// TIA Portal V17 export
// export: Created 2024-01-30T08:49:12.6809505Z, ExportSetting WithDefaults, DisplayName Totally Integrated Automation Portal, DisplayVersion V17 Update 6, DisplayName TIA Portal Openness, DisplayVersion V17 Update 6, DisplayName TIA Portal Version Control Interface, DisplayVersion V17, DisplayName STEP 7 Professional, DisplayVersion V17 Update 6, DisplayName STEP 7 Safety, DisplayVersion V17 Update 6, DisplayName WinCC Advanced, DisplayVersion V17 Update 6
FUNCTION_BLOCK "MeasTable_SQ"   // FB15, GRAPH
AUTHOR : an38503
VERSION : 0.1
// stored: AcknowledgeErrorsRequired true, AutoNumber true, GraphVersion 6.0, InitialValuesAcquisition false, IsIECCheckEnabled false, LanguageInNetworks FBD, LockOperatingMode false, PermanentILProcessingInMANMode false, SetENOAutomatically false, SkipSteps false, UDAEnableTagReadback false, WithAlarmHandling true
   // inherited from GRAPH_BASE
   VAR
      OFF_SQ_BASE : Bool;
   END_VAR
   VAR_INPUT
      OFF_SQ { ExternalAccessible := 'False'; ExternalVisible := 'False'; ExternalWritable := 'False'} : Bool := false;   // Kette ausschalten
      INIT_SQ { ExternalAccessible := 'False'; ExternalVisible := 'False'; ExternalWritable := 'False'} : Bool := false;   // Kette in Initialzustand versetzen
      ACK_EF { ExternalAccessible := 'False'; ExternalVisible := 'False'; ExternalWritable := 'False'} : Bool := false;   // Alle Fehler und Störungen quittieren
      S_PREV { ExternalAccessible := 'False'; ExternalVisible := 'False'; ExternalWritable := 'False'} : Bool := false;   // Vorherigen Schritt am Parameter S_NO ausgeben
      S_NEXT { ExternalAccessible := 'False'; ExternalVisible := 'False'; ExternalWritable := 'False'} : Bool := false;   // Nächsten Schritt am Parameter S_NO anzeigen
      SW_AUTO { ExternalAccessible := 'False'; ExternalVisible := 'False'; ExternalWritable := 'False'} : Bool := false;   // Automatischer Betrieb
      SW_TAP { ExternalAccessible := 'False'; ExternalVisible := 'False'; ExternalWritable := 'False'} : Bool := false;   // Halbautomatisch/Weiterschalten mit Transition
      SW_TOP { ExternalAccessible := 'False'; ExternalVisible := 'False'; ExternalWritable := 'False'} : Bool := false;   // Halbautomatisch/Ignoriere Transition
      SW_MAN { ExternalAccessible := 'False'; ExternalVisible := 'False'; ExternalWritable := 'False'} : Bool := false;   // Handbetrieb
      S_SEL { ExternalAccessible := 'False'; ExternalVisible := 'False'; ExternalWritable := 'False'} : Int := 0;   // Schritt auswählen, der an S_NO ausgegeben werden soll
      S_ON { ExternalAccessible := 'False'; ExternalVisible := 'False'; ExternalWritable := 'False'} : Bool := false;   // Schritt aktivieren, der an Parameter S_NO anliegt
      S_OFF { ExternalAccessible := 'False'; ExternalVisible := 'False'; ExternalWritable := 'False'} : Bool := false;   // Schritt deaktivieren, der an Parameter S_NO anliegt
      T_PUSH { ExternalAccessible := 'False'; ExternalVisible := 'False'; ExternalWritable := 'False'} : Bool := false;   // Schaltfreigabe für Transition im halbautomatischen Betrieb
   END_VAR
   VAR_OUTPUT
      S_NO { ExternalAccessible := 'False'; ExternalVisible := 'False'; ExternalWritable := 'False'} : Int := 0;   // Schrittnummer
      S_MORE { ExternalAccessible := 'False'; ExternalVisible := 'False'; ExternalWritable := 'False'} : Bool := false;   // Weitere Schritte sind vorhanden und können in S_NO angezeigt werden.
      S_ACTIVE { ExternalAccessible := 'False'; ExternalVisible := 'False'; ExternalWritable := 'False'} : Bool := false;   // Schritt, der an Parameter S_NO angezeigt wird, ist aktiv
      ERR_FLT { ExternalAccessible := 'False'; ExternalVisible := 'False'; ExternalWritable := 'False'} : Bool := false;   // Sammelfehler Interlock oder Supervision
      AUTO_ON { ExternalAccessible := 'False'; ExternalVisible := 'False'; ExternalWritable := 'False'} : Bool := false;   // Automatischer Betrieb eingeschaltet
      TAP_ON { ExternalAccessible := 'False'; ExternalVisible := 'False'; ExternalWritable := 'False'} : Bool := false;   // Halbautomatischer Betrieb/Schritt mit Transition eingeschaltet
      TOP_ON { ExternalAccessible := 'False'; ExternalVisible := 'False'; ExternalWritable := 'False'} : Bool := false;   // Halbautomatischer Betrieb/Ignoriere Transition eingeschaltet
      MAN_ON { ExternalAccessible := 'False'; ExternalVisible := 'False'; ExternalWritable := 'False'} : Bool := false;   // Handbetrieb eingeschaltet
   END_VAR
   VAR
      SQ_ProgramRequest { S7_SetPoint := 'True'} : Bool;
      DataHasRead_1 : Bool;
   END_VAR
BEGIN
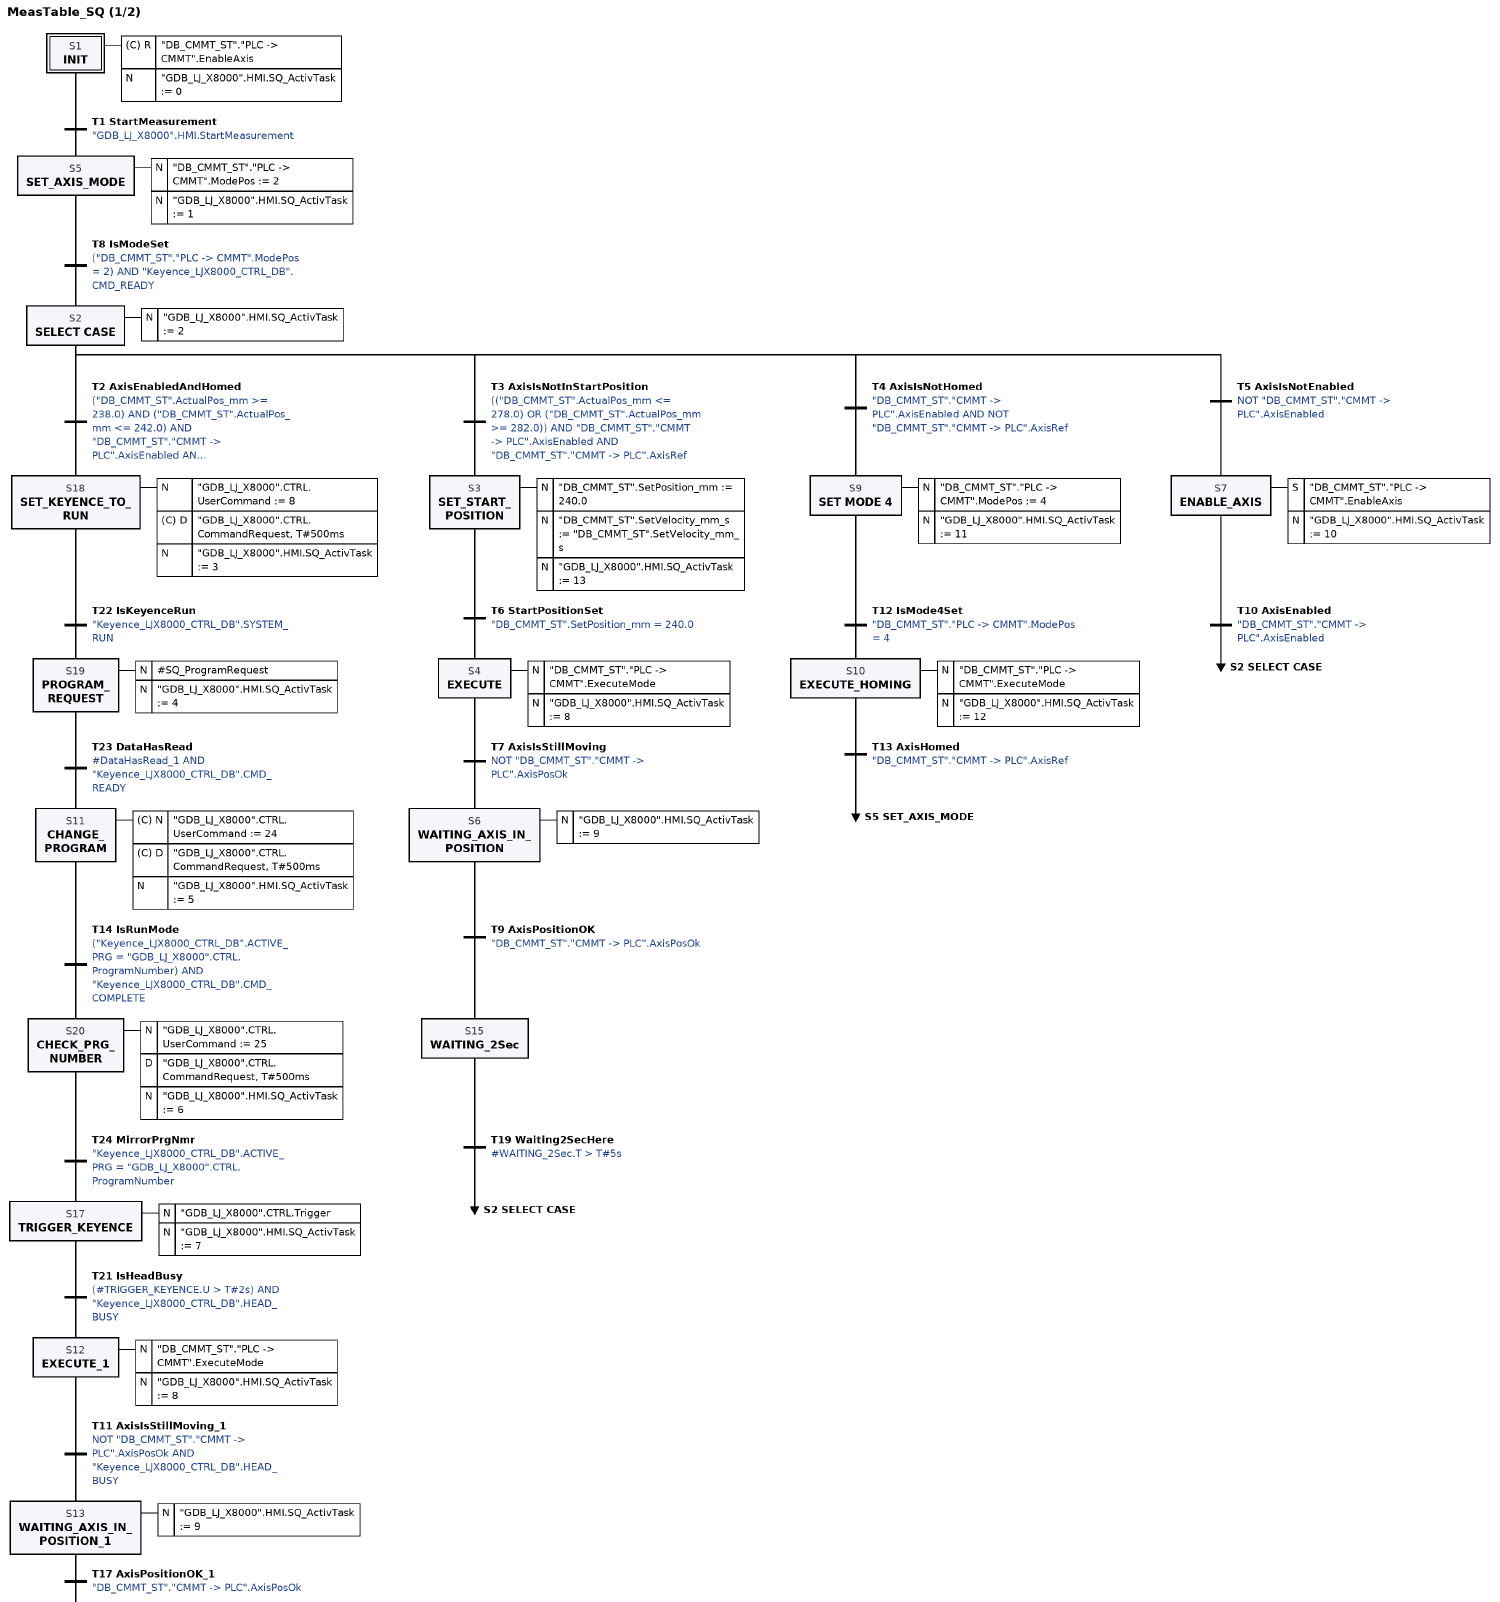
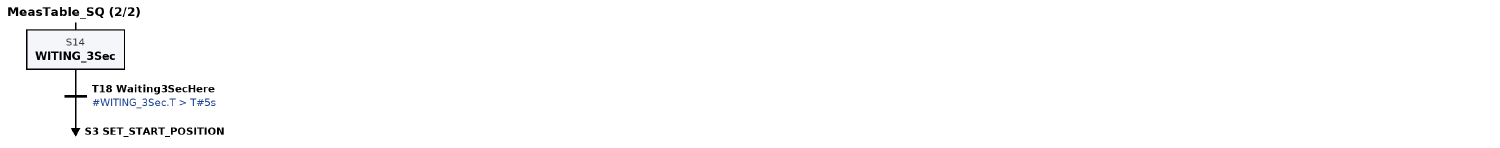
   // sequencer 1
   INITIAL_STEP INIT:   // S1, max time T#10S, warning time T#7S
      interlock C := "GDB_LJ_X8000".HMI.MeasurementMode AND NOT "GDB_LJ_X8000".HMI.HandMode;
      (C)     R    "DB_CMMT_ST"."PLC -> CMMT".EnableAxis
              N    "GDB_LJ_X8000".HMI.SQ_ActivTask := 0
   END_STEP
   TRANSITION StartMeasurement FROM INIT TO SET_AXIS_MODE   // T1
      := "GDB_LJ_X8000".HMI.StartMeasurement;
   END_TRANSITION
   STEP "SELECT CASE":   // S2, max time T#10S, warning time T#7S
              N    "GDB_LJ_X8000".HMI.SQ_ActivTask := 2
   END_STEP
   TRANSITION AxisEnabledAndHomed FROM "SELECT CASE" TO SET_KEYENCE_TO_RUN   // T2
      := ("DB_CMMT_ST".ActualPos_mm >= 238.0) AND ("DB_CMMT_ST".ActualPos_mm <= 242.0) AND "DB_CMMT_ST"."CMMT -> PLC".AxisEnabled AND "DB_CMMT_ST"."CMMT -> PLC".AxisRef AND "Keyence_LJX8000_CTRL_DB".CMD_READY;
   END_TRANSITION
   TRANSITION AxisIsNotInStartPosition FROM "SELECT CASE" TO SET_START_POSITION   // T3
      := (("DB_CMMT_ST".ActualPos_mm <= 278.0) OR ("DB_CMMT_ST".ActualPos_mm >= 282.0)) AND "DB_CMMT_ST"."CMMT -> PLC".AxisEnabled AND "DB_CMMT_ST"."CMMT -> PLC".AxisRef;
   END_TRANSITION
   TRANSITION AxisIsNotHomed FROM "SELECT CASE" TO "SET MODE 4"   // T4
      := "DB_CMMT_ST"."CMMT -> PLC".AxisEnabled AND NOT "DB_CMMT_ST"."CMMT -> PLC".AxisRef;
   END_TRANSITION
   TRANSITION AxisIsNotEnabled FROM "SELECT CASE" TO ENABLE_AXIS   // T5
      := NOT "DB_CMMT_ST"."CMMT -> PLC".AxisEnabled;
   END_TRANSITION
   STEP SET_START_POSITION:   // S3, max time T#10S, warning time T#7S
              N    "DB_CMMT_ST".SetPosition_mm := 240.0
              N    "DB_CMMT_ST".SetVelocity_mm_s := "DB_CMMT_ST".SetVelocity_mm_s
              N    "GDB_LJ_X8000".HMI.SQ_ActivTask := 13
   END_STEP
   TRANSITION StartPositionSet FROM SET_START_POSITION TO EXECUTE   // T6
      := "DB_CMMT_ST".SetPosition_mm = 240.0;
   END_TRANSITION
   STEP EXECUTE:   // S4, max time T#10S, warning time T#7S
              N    "DB_CMMT_ST"."PLC -> CMMT".ExecuteMode
              N    "GDB_LJ_X8000".HMI.SQ_ActivTask := 8
   END_STEP
   TRANSITION AxisIsStillMoving FROM EXECUTE TO WAITING_AXIS_IN_POSITION   // T7
      := NOT "DB_CMMT_ST"."CMMT -> PLC".AxisPosOk;
   END_TRANSITION
   STEP SET_AXIS_MODE:   // S5, max time T#10S, warning time T#7S
              N    "DB_CMMT_ST"."PLC -> CMMT".ModePos := 2
              N    "GDB_LJ_X8000".HMI.SQ_ActivTask := 1
   END_STEP
   TRANSITION IsModeSet FROM SET_AXIS_MODE TO "SELECT CASE"   // T8
      := ("DB_CMMT_ST"."PLC -> CMMT".ModePos = 2) AND "Keyence_LJX8000_CTRL_DB".CMD_READY;
   END_TRANSITION
   STEP WAITING_AXIS_IN_POSITION:   // S6, max time T#10S, warning time T#7S
              N    "GDB_LJ_X8000".HMI.SQ_ActivTask := 9
   END_STEP
   TRANSITION AxisPositionOK FROM WAITING_AXIS_IN_POSITION TO WAITING_2Sec   // T9
      := "DB_CMMT_ST"."CMMT -> PLC".AxisPosOk;
   END_TRANSITION
   STEP ENABLE_AXIS:   // S7, max time T#10S, warning time T#7S
              S    "DB_CMMT_ST"."PLC -> CMMT".EnableAxis
              N    "GDB_LJ_X8000".HMI.SQ_ActivTask := 10
   END_STEP
   TRANSITION AxisEnabled FROM ENABLE_AXIS TO "SELECT CASE"   // T10, jump
      := "DB_CMMT_ST"."CMMT -> PLC".AxisEnabled;
   END_TRANSITION
   STEP "SET MODE 4":   // S9, max time T#10S, warning time T#7S
              N    "DB_CMMT_ST"."PLC -> CMMT".ModePos := 4
              N    "GDB_LJ_X8000".HMI.SQ_ActivTask := 11
   END_STEP
   TRANSITION IsMode4Set FROM "SET MODE 4" TO EXECUTE_HOMING   // T12
      := "DB_CMMT_ST"."PLC -> CMMT".ModePos = 4;
   END_TRANSITION
   STEP EXECUTE_HOMING:   // S10, max time T#10S, warning time T#7S
              N    "DB_CMMT_ST"."PLC -> CMMT".ExecuteMode
              N    "GDB_LJ_X8000".HMI.SQ_ActivTask := 12
   END_STEP
   TRANSITION AxisHomed FROM EXECUTE_HOMING TO SET_AXIS_MODE   // T13, jump
      := "DB_CMMT_ST"."CMMT -> PLC".AxisRef;
   END_TRANSITION
   STEP CHANGE_PROGRAM:   // S11, max time T#10S, warning time T#7S
      (C)     N    "GDB_LJ_X8000".CTRL.UserCommand := 24
      (C)     D    "GDB_LJ_X8000".CTRL.CommandRequest, T#500ms
              N    "GDB_LJ_X8000".HMI.SQ_ActivTask := 5
   END_STEP
   TRANSITION IsRunMode FROM CHANGE_PROGRAM TO CHECK_PRG_NUMBER   // T14
      := ("Keyence_LJX8000_CTRL_DB".ACTIVE_PRG = "GDB_LJ_X8000".CTRL.ProgramNumber) AND "Keyence_LJX8000_CTRL_DB".CMD_COMPLETE;
   END_TRANSITION
   STEP TRIGGER_KEYENCE:   // S17, max time T#10S, warning time T#7S
              N    "GDB_LJ_X8000".CTRL.Trigger
              N    "GDB_LJ_X8000".HMI.SQ_ActivTask := 7
   END_STEP
   TRANSITION IsHeadBusy FROM TRIGGER_KEYENCE TO EXECUTE_1   // T21
      := (#TRIGGER_KEYENCE.U > T#2s) AND "Keyence_LJX8000_CTRL_DB".HEAD_BUSY;
   END_TRANSITION
   STEP EXECUTE_1:   // S12, max time T#10S, warning time T#7S
              N    "DB_CMMT_ST"."PLC -> CMMT".ExecuteMode
              N    "GDB_LJ_X8000".HMI.SQ_ActivTask := 8
   END_STEP
   TRANSITION AxisIsStillMoving_1 FROM EXECUTE_1 TO WAITING_AXIS_IN_POSITION_1   // T11
      := NOT "DB_CMMT_ST"."CMMT -> PLC".AxisPosOk AND "Keyence_LJX8000_CTRL_DB".HEAD_BUSY;
   END_TRANSITION
   STEP WITING_3Sec:   // S14, max time T#10S, warning time T#7S
   END_STEP
   TRANSITION Waiting3SecHere FROM WITING_3Sec TO SET_START_POSITION   // T18, jump
      := #WITING_3Sec.T > T#5s;
   END_TRANSITION
   STEP WAITING_AXIS_IN_POSITION_1:   // S13, max time T#10S, warning time T#7S
              N    "GDB_LJ_X8000".HMI.SQ_ActivTask := 9
   END_STEP
   TRANSITION AxisPositionOK_1 FROM WAITING_AXIS_IN_POSITION_1 TO WITING_3Sec   // T17
      := "DB_CMMT_ST"."CMMT -> PLC".AxisPosOk;
   END_TRANSITION
   STEP WAITING_2Sec:   // S15, max time T#10S, warning time T#7S
   END_STEP
   TRANSITION Waiting2SecHere FROM WAITING_2Sec TO "SELECT CASE"   // T19, jump
      := #WAITING_2Sec.T > T#5s;
   END_TRANSITION
   STEP SET_KEYENCE_TO_RUN:   // S18, max time T#10S, warning time T#7S
      interlock C := NOT "Keyence_LJX8000_CTRL_DB".SYSTEM_RUN;
              N    "GDB_LJ_X8000".CTRL.UserCommand := 8
      (C)     D    "GDB_LJ_X8000".CTRL.CommandRequest, T#500ms
              N    "GDB_LJ_X8000".HMI.SQ_ActivTask := 3
   END_STEP
   TRANSITION IsKeyenceRun FROM SET_KEYENCE_TO_RUN TO PROGRAM_REQUEST   // T22
      := "Keyence_LJX8000_CTRL_DB".SYSTEM_RUN;
   END_TRANSITION
   STEP PROGRAM_REQUEST:   // S19, max time T#10S, warning time T#7S
              N    #SQ_ProgramRequest
              N    "GDB_LJ_X8000".HMI.SQ_ActivTask := 4
   END_STEP
   TRANSITION DataHasRead FROM PROGRAM_REQUEST TO CHANGE_PROGRAM   // T23
      := #DataHasRead_1 AND "Keyence_LJX8000_CTRL_DB".CMD_READY;
   END_TRANSITION
   STEP CHECK_PRG_NUMBER:   // S20, max time T#10S, warning time T#7S
              N    "GDB_LJ_X8000".CTRL.UserCommand := 25
              D    "GDB_LJ_X8000".CTRL.CommandRequest, T#500ms
              N    "GDB_LJ_X8000".HMI.SQ_ActivTask := 6
   END_STEP
   TRANSITION MirrorPrgNmr FROM CHECK_PRG_NUMBER TO TRIGGER_KEYENCE   // T24
      := "Keyence_LJX8000_CTRL_DB".ACTIVE_PRG = "GDB_LJ_X8000".CTRL.ProgramNumber;
   END_TRANSITION
END_FUNCTION_BLOCK
